(* IEC 61131-3 sources: AXOpen/src/components.robotics/app/src/Documentation, 3 files *)

(* ---- Component_1.st ---- *)
USING AXOpen.Core;
{S7.extern=ReadWrite}
CLASS Component_1 EXTENDS AXOpen.Core.AxoObject
    //<ComponentDeclaration>
    VAR PUBLIC
        ExampleCylinder : AXOpen.Components.Robotics.ExampleCylinder;
    END_VAR
    //</ComponentDeclaration>

    //<InitializationArgumentsDeclaration>
    VAR PUBLIC
        _homeSensor : BOOL;
        _workSensor : BOOL;
        _moveHomeSignal : BOOL;
        _moveWorkSignal : BOOL;
    END_VAR
    //</InitializationArgumentsDeclaration>

    METHOD PUBLIC Run
        VAR_INPUT
            parent : IAxoContext;
        END_VAR

        THIS.Initialize(parent);

        //<Initialization>
        ExampleCylinder.Run(THIS, _homeSensor, _workSensor, _moveHomeSignal, _moveWorkSignal);
        //</Initialization>

       THIS.UseInSequencer();
    END_METHOD

    //<Usage>
    VAR PUBLIC
        Sequencer : AxoSequencer;
        Steps : ARRAY[0..3] OF AXOpen.Core.AxoStep;
    END_VAR

    METHOD PRIVATE UseInSequencer

        Sequencer.Initialize(THIS);
        Sequencer.Open();

        IF(Steps[0].Execute(Sequencer, 'Move to home position')) THEN
            IF(ExampleCylinder.MoveToHome.Invoke().IsDone()) THEN
                Sequencer.MoveNext();
            END_IF;
        END_IF;

        IF(Steps[1].Execute(Sequencer, 'Move to work position')) THEN
            IF(ExampleCylinder.MoveToWork.Invoke().IsDone()) THEN
                Sequencer.MoveNext();
            END_IF;
        END_IF;
    END_METHOD

    //</Usage>
END_CLASS

(* ---- Component_2.st ---- *)
USING AXOpen.Core;
{S7.extern=ReadWrite}
CLASS Component_2 EXTENDS AXOpen.Core.AxoObject
    //<ComponentDeclaration>
    VAR PUBLIC
        ExampleCylinder : AXOpen.Components.Robotics.ExampleCylinder;
    END_VAR
    //</ComponentDeclaration>

    //<InitializationArgumentsDeclaration>
    VAR PUBLIC
        _homeSensor : BOOL;
        _workSensor : BOOL;
        _moveHomeSignal : BOOL;
        _moveWorkSignal : BOOL;
    END_VAR
    //</InitializationArgumentsDeclaration>

    METHOD PUBLIC Run
        VAR_INPUT
            parent : IAxoContext;
        END_VAR

        THIS.Initialize(parent);

        //<Initialization>
        ExampleCylinder.Run(THIS, _homeSensor, _workSensor, _moveHomeSignal, _moveWorkSignal);
        //</Initialization>

       THIS.UseInSequencer();
    END_METHOD

    //<Usage>
    VAR PUBLIC
        Sequencer : AxoSequencer;
        Steps : ARRAY[0..3] OF AXOpen.Core.AxoStep;
    END_VAR

    METHOD PRIVATE UseInSequencer

        Sequencer.Initialize(THIS);
        Sequencer.Open();

        IF(Steps[0].Execute(Sequencer, 'Move to home position')) THEN
            IF(ExampleCylinder.MoveToHome.Invoke().IsDone()) THEN
                Sequencer.MoveNext();
            END_IF;
        END_IF;

        IF(Steps[1].Execute(Sequencer, 'Move to work position')) THEN
            IF(ExampleCylinder.MoveToWork.Invoke().IsDone()) THEN
                Sequencer.MoveNext();
            END_IF;
        END_IF;
    END_METHOD

    //</Usage>
END_CLASS

(* ---- DocumentationContext.st ---- *)
NAMESPACE AXOpen.Components.Robotics
    {S7.extern=ReadWrite}
    CLASS DocumentationContext EXTENDS AXOpen.Core.AxoContext
        VAR PUBLIC

        END_VAR

        METHOD PROTECTED OVERRIDE Main
            ;
        END_METHOD
    END_CLASS
END_NAMESPACE
